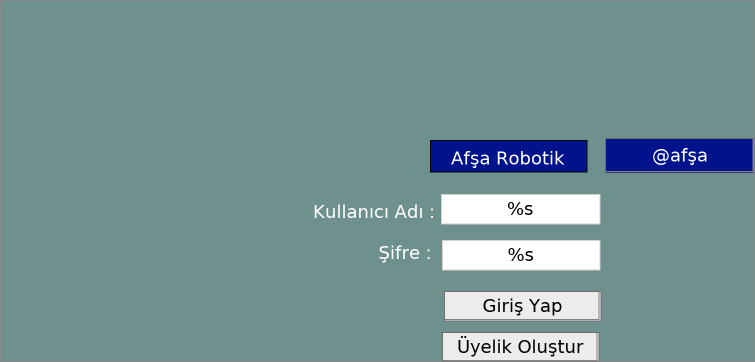
VISUALIZATION Ana_Sayfa  // 755x362
    Rectangle (430,140 157x32)
    Label (299,197 150x30), "Kullanıcı Adı :"
    Label (330,238 150x30), "Şifre :"
    Textfield (441,194 159x30), "%s", text variable: MAIN.kuladi
        OnMouseClick: write the text variable via Edit
    Textfield (442,240 158x30), "%s", text variable: MAIN.sifre
        OnMouseClick: write the text variable via Edit, password
    Button (444,291 157x30), "Giriş Yap"
        tap MAIN.giris
    Button (442,332 157x30), "Üyelik Oluştur"
        tap MAIN.uyelik
        OnMouseClick: change screen: uyelik_sayfa
    Label (288,144 440x29), "Afşa Robotik"
    Button (605,138 150x35), "@afşa", invisible if: MAIN.giris1
        tap MAIN.giris1
        OnMouseClick: change screen: uyelik_sayfa
END_VISUALIZATION

(* stored: Version 1.1.0.1, ProductVersion 3.1.4024.12
   Visu Ana_Sayfa: Id {d926d462-7faf-41ce-beed-cb6fff30f325} *)
